FUNCTION_BLOCK Signal_check
VAR_INPUT
	Signal_IN	:		BOOL;
	T			:		TIME	:=T#2S;
END_VAR
VAR_OUTPUT
	bOK			:		BOOL;
	Signal_OUT  :		BOOL;
END_VAR
VAR
	Signal		:		Signal_generator;
	rtrig		:		R_TRIG;
	timer		:		TON;
END_VAR

Signal(T:=T);
Signal_OUT := Signal.SIGNAL;

rtrig(CLK:= Signal_IN);
timer(IN:=  NOT timer.Q, PT:=2*T);		(* rising edge must 
											be detected during 2 periods TO receive bOK := TRUE *)

END_FUNCTION_BLOCK

(* stored: Version 1.1.0.1, ProductVersion 3.1.4024.16
   POU Signal_check: Id {bc9e2b0e-85d8-4a3b-a4a5-f4378e228aae}, SpecialFunc None *)
